// TIA Portal V20 export
DATA_BLOCK "ET500SP_504"   // DB229
// stored: MemoryReserve 100
   VAR
      "SP504.00 UNWINDER DANCER ENCODER" : Int;
      SPARE1 : Int;
      SPARE2 : Int;
      SPARE3 : Int;
   END_VAR
BEGIN
END_DATA_BLOCK
